(* CoDeSys 2.3 export: CLOCK1S.EXP *)

(* POU clock1s, ST *)
PROGRAM clock1s
VAR
END_VAR
clock1secImpulse:=1;
END_PROGRAM
